{attribute 'GeneratedUsingTerminal: EJ7031-0000-0026'}
{attribute addProperty BoxType "EJ7031-0000-0026"}
{attribute addProperty Id "ControlAT %Q*Control_C948E0F23"}
{attribute addProperty CRC "1519079446"}
{attribute addProperty Size "3"}
TYPE STM_Control_5A8B5016 :
STRUCT
	{attribute addProperty Name "Control"}
	Control AT %Q* : Control_C948E0F2;
END_STRUCT
END_TYPE

(* stored: Version 1.2.0.0, ProductVersion 3.1.4024.9
   DUT STM_Control_5A8B5016: Id {da34c743-c4dd-4d46-a592-404b9536d087} *)
